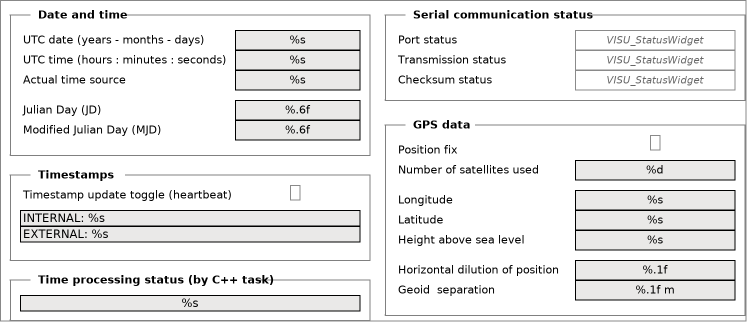
VISUALIZATION VISU_ServicesTimingOverview  // 747x322
VAR_IN_OUT
	ref : ServicesTiming;
    widget : ServicesTimingWidget;
END_VAR
    Polyline (30,280) (10,280) (10,320) (370,320) (370,280) (260,280)
    Polyline (30,15) (10,15) (10,155) (370,155) (370,15) (125,15)
    Polyline (405,125) (385,125) (385,315) (745,315) (745,125) (475,125)
    Rectangle (20,226 340x16), "EXTERNAL: %s", text variable: ref.externalTimestampString
    Rectangle (20,210 340x16), "INTERNAL: %s", text variable: ref.internalTimestampString
    Label (35,5 90x20), "Date and time"
    Label (20,30 200x20), "UTC date (years - months - days)"
    Label (20,50 210x20), "UTC time (hours : minutes : seconds)"
    Label (20,70 195x20), "Actual time source"
    Rectangle (235,70 125x20), "%s", text variable: widget.actualTimeSource
    Rectangle (235,50 125x20), "%s", text variable: ref.utcTimeString
    Rectangle (235,30 125x20), "%s", text variable: ref.utcDateString
    Label (410,5 175x20), "Serial communication status"
    Label (395,160 200x20), "Number of satellites used"
    Label (395,50 200x20), "Transmission status"
    Label (395,30 240x20), "Port status"
    Label (395,260 200x20), "Horizontal dilution of position"
    Label (395,280 200x20), "Geoid separation"
    Label (395,70 235x20), "Checksum status"
    Label (410,115 90x20), "GPS data"
    Label (395,140 200x20), "Position fix"
    Label (35,165 90x20), "Timestamps"
    Frame (575,30 160x20)
        shows VISU_StatusWidget(widget := widget.portHealthStatus)
    Frame (575,50 160x20)
        shows VISU_StatusWidget(widget := widget.transmissionHealthStatus)
    Frame (575,70 160x20)
        shows VISU_StatusWidget(widget := widget.checksumHealthStatus)
    Frame (650,135 10x15)
        shows VISU_State_red_green(state := ref.parts.serialInfo.positionFix)
    Rectangle (575,260 160x20), "%.1f", text variable: ref.parts.serialInfo.horizontalDilutionOfPosition
    Rectangle (575,160 160x20), "%d", text variable: ref.parts.serialInfo.satellitesUsed
    Rectangle (575,280 160x20), "%.1f m", text variable: ref.parts.serialInfo.geoidSeparation
    Frame (290,185 10x15)
        shows VISU_State_gray_green(state := ref.fromEL6688.updateToggle)
    Label (20,185 225x20), "Timestamp update toggle (heartbeat)"
    Polyline (30,175) (10,175) (10,260) (370,260) (370,175) (125,175)
    Polyline (405,15) (385,15) (385,100) (745,100) (745,15) (590,15)
    Rectangle (20,295 340x16), "%s", text variable: widget.errorText
    Label (35,270 225x20), "Time processing status (by C++ task)"
    Rectangle (575,190 160x20), "%s", text variable: widget.longitudeString
    Rectangle (575,210 160x20), "%s", text variable: widget.latitudeString
    Rectangle (575,230 160x20), "%s", text variable: widget.altitudeString
    Label (395,190 200x20), "Longitude"
    Label (395,210 200x20), "Latitude"
    Label (395,230 200x20), "Height above sea level"
    Label (20,100 210x20), "Julian Day (JD)"
    Rectangle (235,100 125x20), "%.6f", text variable: ref.fromCppTiming.utc.mjd + 2400000.5
    Rectangle (235,120 125x20), "%.6f", text variable: ref.fromCppTiming.utc.mjd
    Label (20,120 210x20), "Modified Julian Day (MJD)"
END_VISUALIZATION

(* stored: Version 1.1.0.1, ProductVersion 3.1.4019.2
   Visu VISU_ServicesTimingOverview: Id {b490c1e6-d093-424b-8e86-6ac3f7505684} *)
